FUNCTION_BLOCK FB_CylinderWithPressureFeedback_1 EXTENDS FB_Cylinder
VAR
	_rawPressureValue AT %I* : INT; // Link with analog pressure feedback device
	_statusWord  AT %I* : ST_AnalogSensorStatusWord; // Link with Analog Status Word;
	_targetPressure : INT;
END_VAR
VAR CONSTANT
	ANALOG_MAX : INT := 32765;
END_VAR

PROPERTY AnalogError : BOOL
GET
AnalogError := _statusWord.Error;
END_GET
END_PROPERTY

PROPERTY AtPressure : BOOL
GET
AtPressure := ( _rawPressureValue >= TargetPressure) OR (AtWork AND _simulate) ;
END_GET
END_PROPERTY

PROPERTY TargetPressure : INT
GET
TargetPressure := _targetPressure;
END_GET
SET
/// Simple value range check for setter
IF TargetPressure > 0 AND TargetPressure < ANALOG_MAX THEN
	_targetPressure := TargetPressure;	
END_IF
END_SET
END_PROPERTY

END_FUNCTION_BLOCK

(* stored: Version 1.1.0.1, ProductVersion 3.1.4024.5
   POU FB_CylinderWithPressureFeedback_1: Id {c8e7c96b-126a-404b-a1c3-300273b169c1}, SpecialFunc None
   Property AnalogError: Id {d589fa9a-9fa4-48e9-b82d-239c3a4cc59f}
   Get Get: Id {64404a6d-8451-468a-b586-7e95c20963aa}
   Property AtPressure: Id {6a9e020e-2d04-4336-9b74-5bc07390762b}
   Get Get: Id {087df8b4-4acf-42db-bf77-248476a782be}
   Property TargetPressure: Id {3d7cc59d-eeb5-4a38-8ac7-a2bb98fd3df2}
   Get Get: Id {af101ce1-976c-464f-b5e8-a64f52db6ab4}
   Set Set: Id {810f07c2-e412-413e-8700-e551b52b745b} *)
